FUNCTION_BLOCK Ansteuerung_Ausgaenge
VAR_INPUT
	Saege_Hoch : BOOL;
	Saege_Runter : BOOL;
	Stammklemmung_Oben_Hoch : BOOL;
	Stammklemmung_Oben_Runter : BOOL;
	Stammklemmung_Unten_Hoch : BOOL;
	Stammklemmung_Unten_Runter : BOOL;
	Saege_EIN: BOOL;
	Zufuehrer_Vor : BOOL;
	Zufuehrer_Rueck : BOOL;
	endl_Zufuehrer_vorne : BOOL;
	endl_Zufuehrer_hinten : BOOL;
	endl_Zufuehrer_Vorpos : BOOL;
	endl_Stammklemmung_Oben_Oben : BOOL;
	endl_Stammklemmung_Oben_Unten : BOOL;
	endl_Stammklemmung_Unten_Oben : BOOL;
	endl_Stammklemmung_Unten_Unten : BOOL;
	endl_Saege_Oben : BOOL;
	endl_Saege_Unten : BOOL;
	kettenschmierung_EIN : BOOL;
	
END_VAR
VAR_OUTPUT
	OUT_Saege_Senken AT %Q* : BOOL;
	OUT_Saege_Heben AT %Q* : BOOL;
	OUT_Stammklemmung_Oben_Hoch AT %Q* : BOOL;
	OUT_Stammklemmung_Oben_Runter AT %Q* : BOOL;
	OUT_Stammklemmung_Unten_Hoch AT %Q* : BOOL;
	OUT_Stammklemmung_Unten_Runter AT %Q* : BOOL;
	OUT_Saege_EIN AT %Q* : BOOL;
	OUT_Zufuehrer_Antrieb_Vor AT %Q* : BOOL;
	OUT_Zufuehrer_Antrieb_Rueck AT %Q* : BOOL;
	OUT_Zufuehrer_Antrieb_Enable AT %Q* : BOOL;
	OUT_Kettenschmierung_EIN AT %Q* : BOOL;
END_VAR
VAR
	Saege : Hydr_Ventil;
	Stammklemmung_Oben : Hydr_Ventil;
	Stammklemmung_unten : Hydr_Ventil;
END_VAR


Saege(
	Funktion_A:= Saege_Hoch AND NOT endl_Saege_Oben, 
	Funktion_B:= Saege_Runter AND NOT endl_Saege_Unten, 
	Andere_Ventile_in_Ruhestellung:= Stammklemmung_Oben.Ruhestellung AND Stammklemmung_unten.Ruhestellung, 
	OUT_Spule_A=> OUT_Saege_Heben, 
	OUT_Spule_B=> OUT_Saege_Senken, 
	Status_Invalide=> , 
	Warte_auf_anderes_Ventil=> );

OUT_Saege_EIN := Saege_EIN;
OUT_Kettenschmierung_EIN := kettenschmierung_EIN;
	
Stammklemmung_Oben(
	Funktion_A:= Stammklemmung_Oben_Hoch AND NOT endl_Stammklemmung_Oben_Oben, 
	Funktion_B:= Stammklemmung_Oben_Runter AND NOT endl_Stammklemmung_Oben_Unten, 
	Andere_Ventile_in_Ruhestellung:= Saege.Ruhestellung AND Stammklemmung_unten.Ruhestellung, 
	OUT_Spule_A=> OUT_Stammklemmung_Oben_Hoch, 
	OUT_Spule_B=> OUT_Stammklemmung_Oben_Runter, 
	Status_Invalide=> , 
	Warte_auf_anderes_Ventil=> );
	
Stammklemmung_unten(
	Funktion_A:= Stammklemmung_Unten_Hoch AND NOT endl_Stammklemmung_Unten_Oben, 
	Funktion_B:= Stammklemmung_Unten_Runter AND NOT endl_Stammklemmung_Unten_Unten, 
	Andere_Ventile_in_Ruhestellung:= Saege.Ruhestellung AND Stammklemmung_Oben.Ruhestellung, 
	OUT_Spule_A=> OUT_Stammklemmung_Unten_Hoch, 
	OUT_Spule_B=> OUT_Stammklemmung_Unten_Runter, 
	Status_Invalide=> ,  
	Warte_auf_anderes_Ventil=> );
	
OUT_Zufuehrer_Antrieb_Vor := Zufuehrer_Vor AND NOT Zufuehrer_Rueck AND NOT endl_Zufuehrer_vorne;
OUT_Zufuehrer_Antrieb_Rueck := Zufuehrer_Rueck AND NOT Zufuehrer_Vor AND NOT endl_Zufuehrer_hinten;
OUT_Zufuehrer_Antrieb_Enable := OUT_Zufuehrer_Antrieb_Vor OR OUT_Zufuehrer_Antrieb_Rueck;

END_FUNCTION_BLOCK

(* stored: Version 1.1.0.1, ProductVersion 3.1.4024.16
   POU Ansteuerung_Ausgaenge: Id {ea79a795-b328-4a33-aa54-2323e17ef219}, SpecialFunc None *)
